TYPE T_CodeGTIN : STRING[20];
END_TYPE

(* stored: Version 1.1.0.1
   DUT T_CodeGTIN: Id {40228a55-c217-425d-b436-a785b4e25a68} *)
